// Mitsubishi GX Works2 project: 0126 실린더레더   PLC: Q03UDV

PROGRAM MAIN
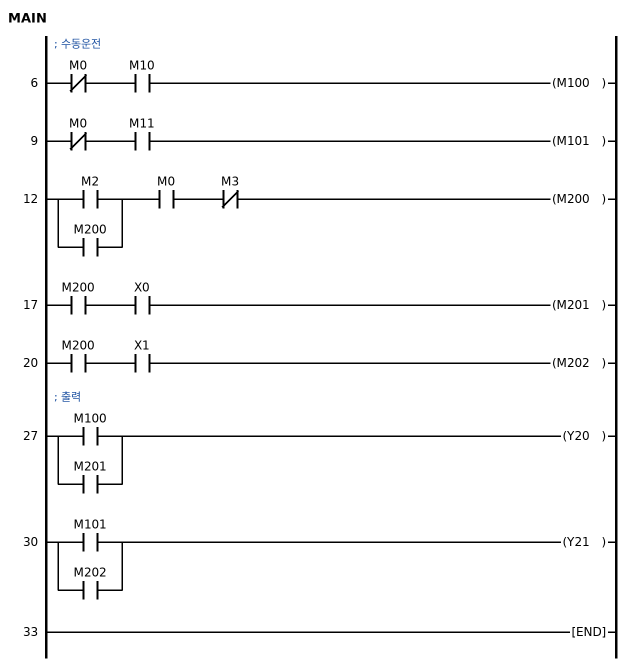
; 수동운전
6     LDI     M0
      AND     M10
      OUT     M100
9     LDI     M0
      AND     M11
      OUT     M101
12    LD      M2
      OR      M200
      AND     M0
      ANI     M3
      OUT     M200
17    LD      M200
      AND     X0
      OUT     M201
20    LD      M200
      AND     X1
      OUT     M202
; 출력
27    LD      M100
      OR      M201
      OUT     Y20
30    LD      M101
      OR      M202
      OUT     Y21
33    END
END_PROGRAM
